// TIA Portal project "IAR-flipm" (V14)

(* hardware
DEVICE "ET 200S station_1"  ET 200S station
   slot 0: "Rack_0"  Rail
   slot 2: "PLC_1"  IM151-8 F-CPU  6ES7 151-8FB00-0AB0  V2.7
      slot 1: "PROFINET interface_1"  PN-IO
         slot 1: "Port_1"  Port
         slot 2: "Port_2"  Port
         slot 3: "Port_3"  Port
   slot 4: "PM-E 24 to 48VDC_1"  PM-E 24 to 48VDC  6ES7 138-4CA50-0AB0
   slot 5: "4DI x 24VDC HF_1"  4DI x 24VDC HF  6ES7 131-4BD01-0AB0
   slot 5: "DP interface_1"  DP  6ES7 138-4HA00-0AB0  V1.0
   slot 6: "4DI x 24VDC HF_2"  4DI x 24VDC HF  6ES7 131-4BD01-0AB0
   slot 7: "4DI x 24VDC HF_3"  4DI x 24VDC HF  6ES7 131-4BD01-0AB0
   slot 8: "4DI x 24VDC HF_4"  4DI x 24VDC HF  6ES7 131-4BD01-0AB0
   slot 9: "4DI x 24VDC HF_5"  4DI x 24VDC HF  6ES7 131-4BD01-0AB0
   slot 10: "2AI x U HF_1"  2AI x U HF  6ES7 134-4LB02-0AB0
   slot 11: "2AI x U HF_2"  2AI x U HF  6ES7 134-4LB02-0AB0
   slot 12: "1 Count 24V_1"  1 COUNT 24V  6ES7 138-4DA04-0AB0  V2.0
   slot 13: "PM-E 24 to 48VDC_2"  PM-E 24 to 48VDC  6ES7 138-4CA50-0AB0
   slot 14: "4DO x 24VDC / 0.5A ST_1"  4DO x 24VDC / 0.5A ST  6ES7 132-4BD02-0AA0
   slot 15: "4DO x 24VDC / 0.5A ST_2"  4DO x 24VDC / 0.5A ST  6ES7 132-4BD02-0AA0
   slot 16: "4DO x 24VDC / 0.5A ST_3"  4DO x 24VDC / 0.5A ST  6ES7 132-4BD02-0AA0
   slot 17: "4DO x 24VDC / 0.5A ST_4"  4DO x 24VDC / 0.5A ST  6ES7 132-4BD02-0AA0
   slot 18: "4DO x 24VDC / 0.5A ST_5"  4DO x 24VDC / 0.5A ST  6ES7 132-4BD02-0AA0
   slot 19: "2AO x U HF_1"  2AO x U HF  6ES7 135-4LB02-0AB0
   slot 20: "2RO x NO/NC 24/230V / 5A_1"  2RO x NO/NC 24/230V / 5A  6ES7 132-4HB50-0AB0
*)

// ===== PLC "PLC_1"  IM151-8 F-CPU =====

VAR_GLOBAL   // PLC tag table "Default tag table"
   "ButtonStart" AT %I1.0 : Bool;
   "ButtonStop" AT %I1.1 : Bool;   // signal inverted
   "SwitchAuto/Man" AT %I1.2 : Bool;
   "ButtonReset" AT %I1.3 : Bool;
   "SensorDetectionLeft" AT %I2.0 : Bool;   // signal inverted
   "SensorDetectionRight" AT %I2.2 : Bool;   // signal inverted
   "EmergencyStop" AT %I2.3 : Bool;   // signal inverted
   "SensorGripperUp" AT %I3.0 : Bool;
   "SensorGripperDown" AT %I3.1 : Bool;
   "SensorGripperOpen" AT %I3.2 : Bool;
   "SensorGripperClose" AT %I3.3 : Bool;
   "SensorGripperTurnCW" AT %I4.0 : Bool;
   "SensorGripperTurnCCW" AT %I4.1 : Bool;
   "SensorDetectionCenter" AT %I4.3 : Bool;   // signal inverted
   "LigthButtonStart" AT %Q11.0 : Bool;
   "LightButtonReset" AT %Q11.1 : Bool;
   "LightQ1" AT %Q11.2 : Bool;
   "LightQ2" AT %Q11.3 : Bool;
   "Conveyor CW" AT %Q12.0 : Bool;
   "Conveyor CCW" AT %Q12.1 : Bool;
   "ReduceCoveyorSpeed" AT %Q12.2 : Bool;
   "GripperUp" AT %Q13.0 : Bool;
   "GripperDown" AT %Q13.1 : Bool;
   "GripperOpen" AT %Q13.2 : Bool;
   "GripperClose" AT %Q13.3 : Bool;
   "GripperTurnCCW" AT %Q14.0 : Bool;
   "GripperTurnCW" AT %Q14.1 : Bool;
   "TotalObjects" AT %MW0 : Int;
END_VAR

FUNCTION "Init" : Void   // FC1, SCL
{ S7_Optimized_Access := 'FALSE' }
VERSION : 0.1
   VAR_INPUT
      Sensor_Gripper_UP : Bool;
      Sensor_Gripper_TurnCCW : Bool;
      Button_Start : Bool;
      Sensor_Gripper_Open : Bool;
   END_VAR
   VAR_OUTPUT
      Gripper_TurnCW : Bool;
      Gripper_down : Bool;
      Gripper_Close : Bool;
      Gripper_UP : Bool;
      Gripper_TurnCCW : Bool;
      Gripper_Open : Bool;
   END_VAR
   VAR_IN_OUT
      State : Int;
      TotalObject : Int;
   END_VAR
BEGIN
   CASE #State OF
       0:
           IF #Button_Start THEN
               #State := 1;
           END_IF;
       1:
           #Gripper_Close := FALSE;
           #Gripper_down := FALSE;
           #Gripper_Open := FALSE;
           #Gripper_UP := TRUE;
           IF #Sensor_Gripper_UP = TRUE THEN
               #State := 2;
           END_IF;
       2:
           #Gripper_TurnCCW := TRUE;
           IF #Sensor_Gripper_TurnCCW = TRUE THEN
               #State := 3;
           END_IF;
       3:
           #Gripper_Open := TRUE;
           IF #Sensor_Gripper_UP THEN
               #State := 4;
               #TotalObject := 0;
           END_IF;
   END_CASE;
END_FUNCTION

FUNCTION "Idle" : Void   // FC2, SCL
{ S7_Optimized_Access := 'FALSE' }
VERSION : 0.1
   VAR_INPUT
      Sensor_detection_right : Bool;
      Sensor_detection_left : Bool;
      Sensor_detection_mid : Bool;
      Clearence : Bool;
   END_VAR
   VAR_OUTPUT
      Conveyor_CW : Bool;
   END_VAR
   VAR_IN_OUT
      State : Int;
      TotalObjects : Int;
   END_VAR
   VAR_TEMP
      seen : Bool;
      gezien : Bool;
   END_VAR
BEGIN
   CASE #State OF
       4:
           IF #Sensor_detection_left = FALSE  THEN
               #Conveyor_CW := TRUE;
               #State := 5;
               #TotalObjects := #TotalObjects + 1;
           END_IF;

           IF #Sensor_detection_mid = FALSE THEN
               #State := 7;
           END_IF;

           IF #Sensor_detection_right = FALSE THEN

               IF #Clearence = FALSE THEN

               #State := 6;
           END_IF;

       5:
           IF #Sensor_detection_left = TRUE THEN
               #State := 4;
           END_IF;
       6:
           #Conveyor_CW := FALSE;
           IF #Sensor_detection_right = TRUE OR #Clearence = TRUE THEN
               #State := 4;
               #Conveyor_CW := TRUE;
           END_IF;
   END_CASE;
END_FUNCTION

FUNCTION "Execute" : Void   // FC3, SCL
{ S7_Optimized_Access := 'FALSE' }
VERSION : 0.1
   VAR_INPUT
      Sensor_Detection_Mid : Bool;
      Sensor_Gripper_Open : Bool;
      Sensor_Gripper_TurnCCW : Bool;
      Sensor_Gripper_UP : Bool;
      Sensor_Gripper_Close : Bool;
      Sensor_Gripper_TurnCW : Bool;
      Sensor_Gripper_Down : Bool;
      Sensor_Conveyor_Right : Bool;
      Clearence : Bool;
   END_VAR
   VAR_OUTPUT
      Gripper_TurnCW : Bool;
      Gripper_down : Bool;
      Gripper_Close : Bool;
      Gripper_UP : Bool;
      Gripper_TurnCCW : Bool;
      Gripper_Open : Bool;
      Conveyor_CW : Bool;
      Conveyor_CCW : Bool;
      Conveyor_Speed_Slow : Bool;
   END_VAR
   VAR_IN_OUT
      State : Int;
   END_VAR
   VAR_TEMP
      Turned_CCW : Bool;
      Turn : Int;
   END_VAR
BEGIN
   CASE #State OF
       7:
           #Conveyor_CW := FALSE;
           #Conveyor_Speed_Slow := TRUE;
           #Conveyor_CCW := TRUE;
           #State := 8;
       8:
           IF #Sensor_Detection_Mid = TRUE THEN
               #Conveyor_CCW := FALSE;
               #Conveyor_Speed_Slow := FALSE;
               #State := 9;
           END_IF;
       9:
           #Gripper_UP := FALSE;
           #Gripper_down := TRUE;
           IF #Sensor_Gripper_Down = TRUE THEN
               #State := 10;
           END_IF;
       10:
           #Gripper_Open := FALSE;
           #Gripper_Close := TRUE;
           IF #Sensor_Gripper_Close = TRUE THEN
               #State := 11;
           END_IF;
       11:
           #Gripper_down := FALSE;
           #Gripper_UP := TRUE;
           IF #Sensor_Gripper_UP = TRUE THEN
               #State := 12;
           END_IF;
       12:
           IF #Sensor_Gripper_TurnCCW = TRUE THEN
               #State := 13;
           END_IF;
           IF #Sensor_Gripper_TurnCW = TRUE THEN
               #State := 14;
           END_IF;
       13:
           #Gripper_TurnCCW := FALSE;
           #Gripper_TurnCW := TRUE;
           IF #Sensor_Gripper_TurnCW = TRUE THEN
               #State := 15;
           END_IF;
       14:
           #Gripper_TurnCW := FALSE;
           #Gripper_TurnCCW := TRUE;
           IF #Sensor_Gripper_TurnCCW = TRUE THEN
               #State := 15;
           END_IF;
       15:
           #Gripper_UP := FALSE;
           #Gripper_down := TRUE;
           IF #Sensor_Gripper_Down = TRUE THEN
               #State := 16;
           END_IF;
       16:
           #Gripper_Close := FALSE;
           #Gripper_Open := true;
           IF #Sensor_Gripper_Open = TRUE THEN
               #State := 17;
           END_IF;
       17:
           #Gripper_down := FALSE;
           #Gripper_UP := TRUE;
           IF #Sensor_Gripper_UP = TRUE THEN
               #State := 18;
           END_IF;
       18:
           IF #Sensor_Conveyor_Right = TRUE OR #Clearence = TRUE THEN
               #Conveyor_CW := TRUE;
               IF #Sensor_Detection_Mid = FALSE THEN
                   #State := 19;
               END_IF;
           ELSE
               #Conveyor_CW := FALSE;
           END_IF;
       19:
           IF #Sensor_Detection_Mid = TRUE THEN
               #State := 4;
           END_IF;

   END_CASE;
END_FUNCTION

ORGANIZATION_BLOCK "Main"   // OB1, SCL
TITLE = "Main Program Sweep (Cycle)"
{ S7_Optimized_Access := 'FALSE' }
VERSION : 0.1
   VAR_TEMP
      OB1_EV_CLASS : Byte;   // Bits 0-3 = 1 (Coming event), Bits 4-7 = 1 (Event class 1)
      OB1_SCAN_1 : Byte;   // 1 (Cold restart scan 1 of OB 1), 3 (Scan 2-n of OB 1)
      OB1_PRIORITY : Byte;   // Priority of OB Execution
      OB1_OB_NUMBR : Byte;   // 1 (Organization block 1, OB1)
      OB1_RESERVED_1 : Byte;   // Reserved for system
      OB1_RESERVED_2 : Byte;   // Reserved for system
      OB1_PREV_CYCLE : Int;   // Cycle time of previous OB1 scan (milliseconds)
      OB1_MIN_CYCLE : Int;   // Minimum cycle time of OB1 (milliseconds)
      OB1_MAX_CYCLE : Int;   // Maximum cycle time of OB1 (milliseconds)
      OB1_DATE_TIME : Date_And_Time;   // Date and time OB1 started
      TotalObjects : Int;
      state : Int;
   END_VAR
BEGIN
   "Init" (
          Sensor_Gripper_UP:="SensorGripperUp",
          Sensor_Gripper_TurnCCW:="SensorGripperTurnCCW",
          Button_Start:="ButtonStart",
          Gripper_down=>"GripperDown",
          Gripper_Close=>"GripperClose",
          Gripper_TurnCW=>"GripperTurnCW",
          Sensor_Gripper_Open:="SensorGripperOpen",
          Gripper_UP=>"GripperUp",
          Gripper_TurnCCW=>"GripperTurnCCW",
          Gripper_Open=>"GripperOpen",
          State:=#state,
           TotalObject:="TotalObjects");


   "Idle"(
          Sensor_detection_right:="SensorDetectionRight",
          Sensor_detection_left:="SensorDetectionLeft",
          Sensor_detection_mid:="SensorDetectionCenter",
          Clearence:="SwitchAuto/Man",
          Conveyor_CW=>"Conveyor CW",
          State:=#state,
          TotalObjects:="TotalObjects");

   "Execute"(
             Sensor_Detection_Mid:="SensorDetectionCenter",
             Sensor_Gripper_Open:="SensorGripperOpen",
             Sensor_Gripper_TurnCCW:="SensorGripperTurnCCW",
             Sensor_Gripper_UP:="SensorGripperUp",
             Sensor_Gripper_Close:="SensorGripperClose",
             Sensor_Gripper_TurnCW:="SensorGripperTurnCW",
             Sensor_Gripper_Down:="SensorGripperDown",
             Sensor_Conveyor_Right:="SensorDetectionRight",
             Clearence:="SwitchAuto/Man",
             Gripper_TurnCW=>"GripperTurnCW",
             Gripper_down=>"GripperDown",
             Gripper_Close=>"GripperClose",
             Gripper_UP=>"GripperUp",
             Gripper_TurnCCW=>"GripperTurnCCW",
             Gripper_Open=>"GripperOpen",
             Conveyor_CW=>"Conveyor CW",
             Conveyor_CCW=>"Conveyor CCW",
             Conveyor_Speed_Slow=>"ReduceCoveyorSpeed",
             State:=#state);
END_ORGANIZATION_BLOCK